{attribute 'qualified_only'}
VAR_GLOBAL
	fbMachineConfiguration		: FB_MachineConfiguration;
	fbHMIConfiguration			: FB_HMIConfiguration;
	
	fbMachineTemplate1			: FB_MachineTemplate1;
	fbMachineTemplate2			: FB_MachineTemplate2;
	fbMachineTemplate3			: FB_MachineTemplate3;
	
END_VAR

(* stored: Version 1.1.0.1, ProductVersion 3.1.4024.15
   GVL GVL_MachineVariable: Id {cd0e9623-7f5e-4ae1-835b-923ddeb15d5b} *)
